// TIA Portal V18 export
FUNCTION_BLOCK "manual_digital"   // FB13, FBD
{ S7_Optimized_Access := 'TRUE' }
VERSION : 0.1
// stored: AutoNumber true, IsIECCheckEnabled false, IsRetainMemResEnabled false, MemoryReserve 100, SetENOAutomatically false, UDAEnableTagReadback false
   VAR_INPUT
      ALLOWED : Bool;
      xFwdOk : Bool;
      xRevOk : Bool;
      xFwdFastOK : Bool;
      xRevFastOK : Bool;
   END_VAR
   VAR_OUTPUT
      FWD : Bool;
      REV : Bool;
      FAST : Bool;
   END_VAR
   VAR_IN_OUT
      btn_FWD : Bool;
      btn_REV : Bool;
   END_VAR
   VAR
      lbs { S7_SetPoint := 'True'} : "last_button_stands";
      ton_quick { S7_SetPoint := 'True'} : TON_TIME;
   END_VAR
BEGIN

REGION Network 1
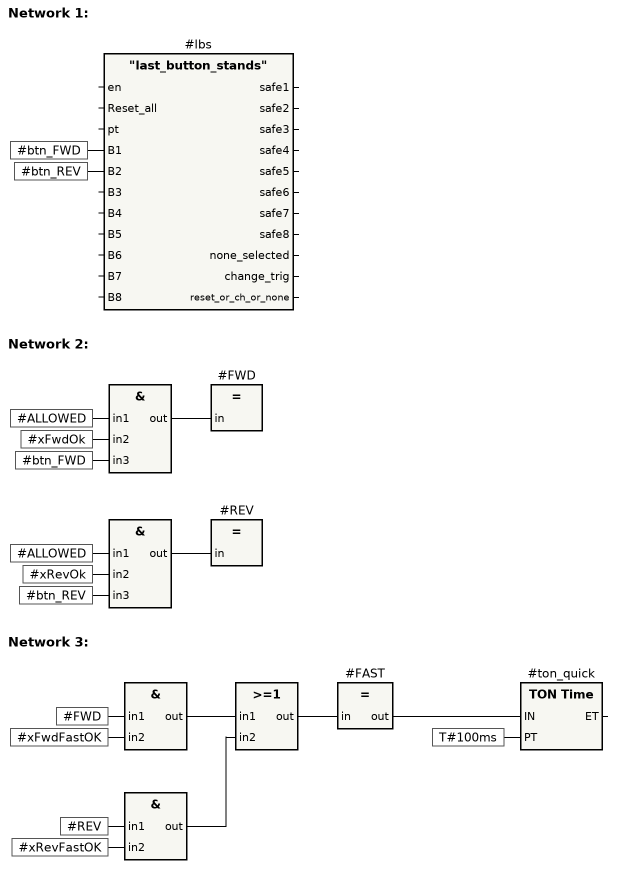
   #lbs(B1 := #btn_FWD, B2 := #btn_REV);   // "last_button_stands"
END_REGION

REGION Network 2
   #FWD := #ALLOWED AND #xFwdOk AND #btn_FWD;
   #REV := #ALLOWED AND #xRevOk AND #btn_REV;
END_REGION

REGION Network 3
   #FAST := (#FWD AND #xFwdFastOK) OR (#REV AND #xRevFastOK);
   #ton_quick(IN := #FAST, PT := T#100ms);   // TON
END_REGION
END_FUNCTION_BLOCK
